{attribute addProperty BoxType "KL9900-0062"}
{attribute addProperty Id "Channel_1Channel_D761A7C100"}
{attribute addProperty CRC "2446581870"}
{attribute addProperty SizeInBites "0"}
{attribute addProperty SizeInBytes "0"}
TYPE KL_91D3E06E :
STRUCT
	{attribute addProperty Name "Channel_1"}
	Channel_1 : Channel_D761A7C1;
END_STRUCT
END_TYPE

(* stored: Version 1.2.0.0, ProductVersion 3.1.4024.9
   DUT KL_91D3E06E: Id {755a2e26-b859-44b0-be9a-91812a6e93a7} *)
